(* PLC project Test Library, INSA Strasbourg Test Library 1.0, author Mathieu Giamberini *)
(* stored: creationDateTime 2024-10-04T15:34:52, modificationDateTime 2024-11-05T16:23:40 *)

FUNCTION_BLOCK TestBlock1
  VAR
    Test2 : DINT;
  END_VAR
  VAR RETAIN
    Test1 : INT := 0;
  END_VAR
  VAR_OUTPUT
    LED : BOOL := 0;
  END_VAR
  VAR_OUTPUT RETAIN
    ID : BYTE := 160;  (* 0xA0 *)
  END_VAR
  VAR RETAIN
    threashold : INT := 20;
  END_VAR
  VAR
    Test0 : Test;
    BNO0550 : BNO055;
  END_VAR

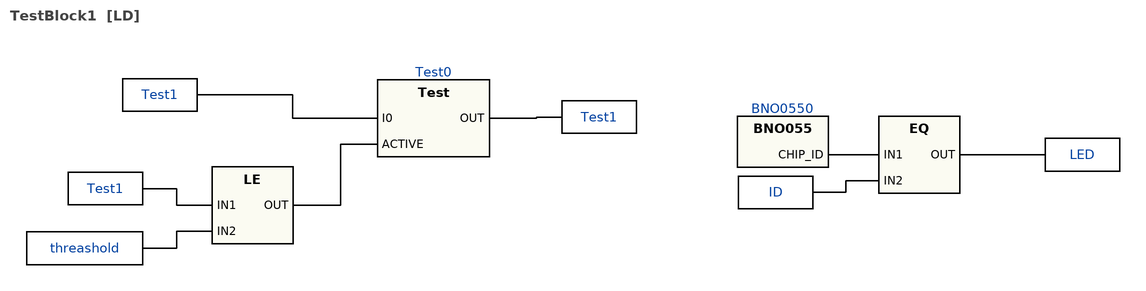
(* LD diagram, written out as Structured Text *)
Test0(I0 := Test1, ACTIVE := Test1 <= threashold);
Test1 := Test0.OUT;
BNO0550();
LED := BNO0550.CHIP_ID = ID;
END_FUNCTION_BLOCK

PROGRAM program0
  VAR
    TestBlock10 : TestBlock1;
    LED : BOOL;
  END_VAR

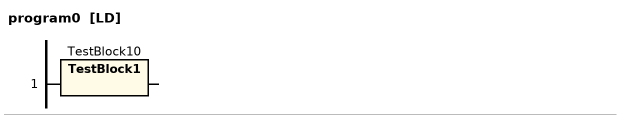
(* LD diagram, written out as Structured Text *)
TestBlock10();
END_PROGRAM

CONFIGURATION Config0
  RESOURCE Res0 ON PLC
    TASK task0(INTERVAL := T#20ms, PRIORITY := 0);
    PROGRAM instance0 WITH task0 : program0;
  END_RESOURCE
END_CONFIGURATION
